INTERFACE I_Subscriber

METHOD Update
VAR_INPUT
	Event : I_Event;
END_VAR
END_METHOD

END_INTERFACE

(* stored: Version 1.1.0.1, ProductVersion 3.1.4024.11
   Itf I_Subscriber: Id {5fe761e5-975d-464e-8146-7a7f983afe21}
   Method Update: Id {a20689a2-3fa1-4532-9bd0-c85a5f69ff3e} *)
